FUNCTION_BLOCK Carriage
  (* Version 1.0, 2007-08-23, Goran Cengic, Chalmers *)
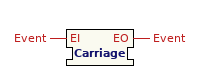
  EVENT_INPUT
    EI;
  END_EVENT
  EVENT_OUTPUT
    EO;
  END_EVENT
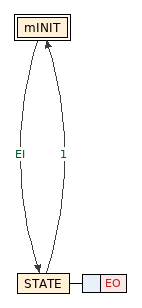
  EC_STATES
    mINIT;
    STATE : -> EO;
  END_STATES
  EC_TRANSITIONS
    mINIT TO STATE := EI;
    STATE TO mINIT := 1;
  END_TRANSITIONS
END_FUNCTION_BLOCK
(* other elements stored in the file *)
(* ECAction Algorithm="GetCarriage" Output="EO"/ *)
(* Algorithm Name="GetCarriage"> <Other Language="Java" Text="System.out.println(&#34;Getting Carriage!&#34;);" /> </Algorithm *)
